{attribute 'GeneratedUsingTerminal: EJ1918-0000-0017'}
{attribute addProperty BoxType "EJ1918-0000-0017"}
{attribute addProperty Id "FSoE_CommandUSINT1FSIN_Module_1_Channel_1_InputBOOL1FSIN_Module_1_Channel_2_InputBOOL1FSIN_Module_1_Module_FaultBOOL1FSIN_Module_2_Channel_1_InputBOOL1FSIN_Module_2_Channel_2_InputBOOL1FSIN_Module_2_Module_FaultBOOL1FSIN_Module_3_Channel_1_InputBOOL1FSIN_Module_3_Channel_2_InputBOOL1FSIN_Module_3_Module_FaultBOOL1FSIN_Module_4_Channel_1_InputBOOL1FSIN_Module_4_Channel_2_InputBOOL1FSIN_Module_4_Module_FaultBOOL1FSoE_CRC_000UINT2FSoE_Connection_IDUINT2"}
{attribute addProperty CRC "2667874397"}
{attribute addProperty Size "17"}
TYPE FSOE_9F04885D :
STRUCT
	{attribute addProperty Name "FSoE_Command"}
	FSoE_Command : USINT;
	{attribute addProperty Name "FSIN_Module_1_Channel_1_Input"}
	FSIN_Module_1_Channel_1_Input : BOOL;
	{attribute addProperty Name "FSIN_Module_1_Channel_2_Input"}
	FSIN_Module_1_Channel_2_Input : BOOL;
	{attribute addProperty Name "FSIN_Module_1_Module_Fault"}
	FSIN_Module_1_Module_Fault : BOOL;
	{attribute addProperty Name "FSIN_Module_2_Channel_1_Input"}
	FSIN_Module_2_Channel_1_Input : BOOL;
	{attribute addProperty Name "FSIN_Module_2_Channel_2_Input"}
	FSIN_Module_2_Channel_2_Input : BOOL;
	{attribute addProperty Name "FSIN_Module_2_Module_Fault"}
	FSIN_Module_2_Module_Fault : BOOL;
	{attribute addProperty Name "FSIN_Module_3_Channel_1_Input"}
	FSIN_Module_3_Channel_1_Input : BOOL;
	{attribute addProperty Name "FSIN_Module_3_Channel_2_Input"}
	FSIN_Module_3_Channel_2_Input : BOOL;
	{attribute addProperty Name "FSIN_Module_3_Module_Fault"}
	FSIN_Module_3_Module_Fault : BOOL;
	{attribute addProperty Name "FSIN_Module_4_Channel_1_Input"}
	FSIN_Module_4_Channel_1_Input : BOOL;
	{attribute addProperty Name "FSIN_Module_4_Channel_2_Input"}
	FSIN_Module_4_Channel_2_Input : BOOL;
	{attribute addProperty Name "FSIN_Module_4_Module_Fault"}
	FSIN_Module_4_Module_Fault : BOOL;
	{attribute addProperty Name "FSoE_CRC_000"}
	FSoE_CRC_000 : UINT;
	{attribute addProperty Name "FSoE_Connection_ID"}
	FSoE_Connection_ID : UINT;
END_STRUCT
END_TYPE

(* stored: Version 1.2.0.0, ProductVersion 3.1.4024.9
   DUT FSOE_9F04885D: Id {fdfe3da3-8034-40a7-b1af-d87aacc818d5} *)
